(* PLC project SafeLOGIC, BrAutomation SafeDESIGNER  5.24.1.0 *)
(* stored: companyURL http://www.br-automation.com, creationDateTime Tue Nov 25 17:09:51 2025 *)

PROGRAM PARA_BOOL

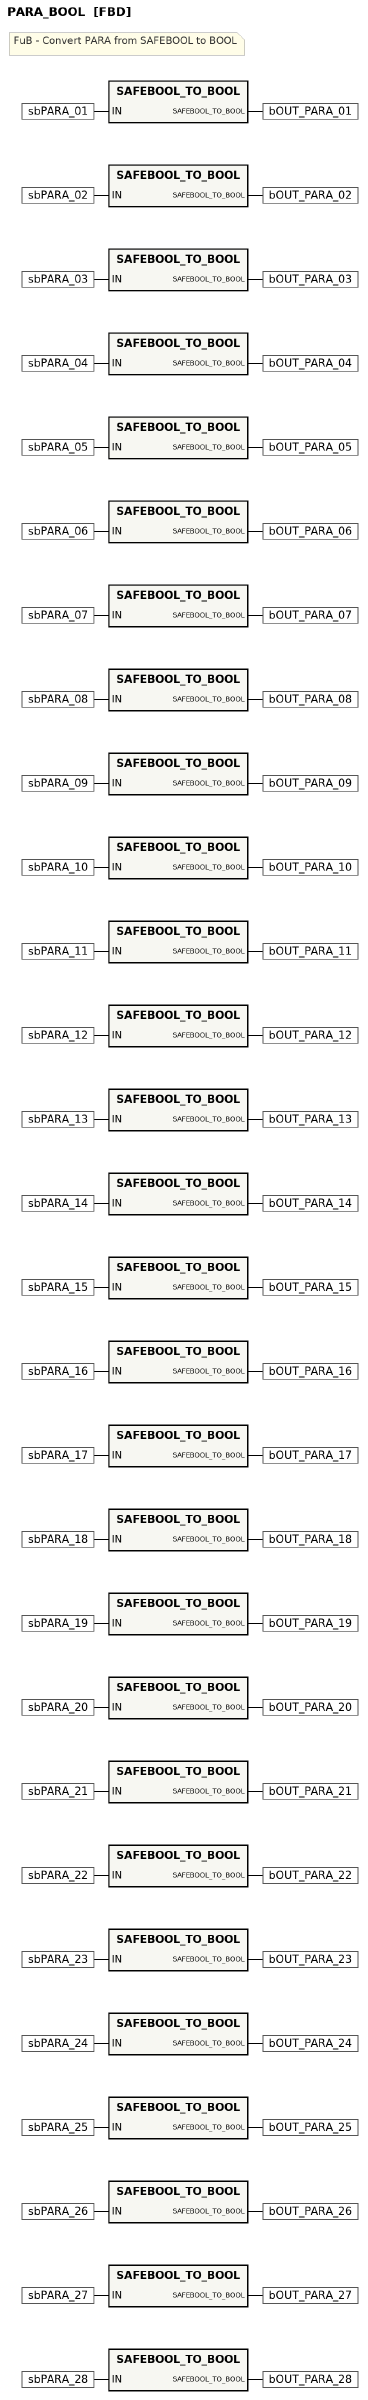
(* FBD diagram, written out as Structured Text *)
(* FuB - Convert PARA from SAFEBOOL to BOOL *)
bOUT_PARA_01 := SAFEBOOL_TO_BOOL(sbPARA_01);
bOUT_PARA_02 := SAFEBOOL_TO_BOOL(sbPARA_02);
bOUT_PARA_03 := SAFEBOOL_TO_BOOL(sbPARA_03);
bOUT_PARA_04 := SAFEBOOL_TO_BOOL(sbPARA_04);
bOUT_PARA_05 := SAFEBOOL_TO_BOOL(sbPARA_05);
bOUT_PARA_06 := SAFEBOOL_TO_BOOL(sbPARA_06);
bOUT_PARA_07 := SAFEBOOL_TO_BOOL(sbPARA_07);
bOUT_PARA_08 := SAFEBOOL_TO_BOOL(sbPARA_08);
bOUT_PARA_09 := SAFEBOOL_TO_BOOL(sbPARA_09);
bOUT_PARA_10 := SAFEBOOL_TO_BOOL(sbPARA_10);
bOUT_PARA_11 := SAFEBOOL_TO_BOOL(sbPARA_11);
bOUT_PARA_12 := SAFEBOOL_TO_BOOL(sbPARA_12);
bOUT_PARA_13 := SAFEBOOL_TO_BOOL(sbPARA_13);
bOUT_PARA_14 := SAFEBOOL_TO_BOOL(sbPARA_14);
bOUT_PARA_15 := SAFEBOOL_TO_BOOL(sbPARA_15);
bOUT_PARA_16 := SAFEBOOL_TO_BOOL(sbPARA_16);
bOUT_PARA_17 := SAFEBOOL_TO_BOOL(sbPARA_17);
bOUT_PARA_18 := SAFEBOOL_TO_BOOL(sbPARA_18);
bOUT_PARA_19 := SAFEBOOL_TO_BOOL(sbPARA_19);
bOUT_PARA_20 := SAFEBOOL_TO_BOOL(sbPARA_20);
bOUT_PARA_21 := SAFEBOOL_TO_BOOL(sbPARA_21);
bOUT_PARA_22 := SAFEBOOL_TO_BOOL(sbPARA_22);
bOUT_PARA_23 := SAFEBOOL_TO_BOOL(sbPARA_23);
bOUT_PARA_24 := SAFEBOOL_TO_BOOL(sbPARA_24);
bOUT_PARA_25 := SAFEBOOL_TO_BOOL(sbPARA_25);
bOUT_PARA_26 := SAFEBOOL_TO_BOOL(sbPARA_26);
bOUT_PARA_27 := SAFEBOOL_TO_BOOL(sbPARA_27);
bOUT_PARA_28 := SAFEBOOL_TO_BOOL(sbPARA_28);
END_PROGRAM
